{attribute 'qualified_only'}
VAR_GLOBAL
    iCompletionHMI : ARRAY[0..CONST.STATION_NUMBER] OF INT;

    lrSpeedMover       : LREAL := 20.0;
    lrAccelMover       : LREAL; // is lrAccelMoverSlider^2
    lrAccelMoverSlider : LREAL := 0.4;
END_VAR

(* stored: Version 1.1.0.1, ProductVersion 3.1.4024.6
   GVL SIMU: Id {345b4519-5ad6-46f0-ab8f-5a823ebcb6f9} *)
